{warning <'Multi will not function for Sectors that span multiple XTS tracks'>}    
FUNCTION_BLOCK FB_SingularTrackSector
VAR_INPUT
	PlanarTrackIndex				: E_TrackNum := E_TrackNum.Small;
END_VAR
VAR_IN_OUT
	refPlanarTracks					: ARRAY[*] OF ST_PlanarTrackConfig; //NOTE ref array is 0-based!
END_VAR                     		
VAR                             	
	InitDone						: BOOL;
	stSectorConfig					: ST_SectorConfig;
	LowerBoundPlanarTrackConfig		: DINT;
	UpperBoundPlanarTrackConfig		: DINT;
	refXtsMover						: Tc3_XTS_Utility.ST_PositionInfo;
	refPlanarMover					: MoverSort;
	stTrackSectorStatus				: ST_SectorStatus;
END_VAR

IF UpperBoundPlanarTrackConfig = 0 THEN
	_M_Init();
ELSE
	InitDone	:= TRUE;
END_IF

IF InitDone THEN
	_M_UpdateSectorStatus();
END_IF

METHOD PRIVATE _M_Init
LowerBoundPlanarTrackConfig	:= LOWER_BOUND(refPlanarTracks,1);
UpperBoundPlanarTrackConfig	:= UPPER_BOUND(refPlanarTracks,1);
END_METHOD

METHOD PROTECTED _M_IsOnPlanarSector : BOOL
//note refPlanarTracks ARRAY is 0-based!
IF ADR(refPlanarTracks[(PlanarTrackIndex-1)]) <> Tc3_Module.NULL THEN
	_M_IsOnPlanarSector	:= (refPlanarMover.TrackID = refPlanarTracks[(PlanarTrackIndex-1)].MCTrack.TrackOID) 
							AND IsBetween(value := refPlanarMover.MoverPos, 
												minV := stSectorConfig.TrackSectorStartPosn, 
												maxV := stSectorConfig.TrackSectorEndPosn);
END_IF
END_METHOD

METHOD PROTECTED _M_IsOnXtsSector : BOOL
_M_IsOnXtsSector	:= ((refXtsMover.nTrackObjectid = stSectorConfig.ObjectId) OR
											(refXtsMover.nPartObjectid = stSectorConfig.ObjectId)) AND
											(IsBetween(value := refXtsMover.fPartPosition, 
											minV := stSectorConfig.PartSectorStartPosn, 
											maxV := stSectorConfig.PartSectorEndPosn) OR
											IsBetween(value := refXtsMover.fTrackPosition, 
											minV := stSectorConfig.TrackSectorStartPosn, 
											maxV := stSectorConfig.TrackSectorEndPosn));
END_METHOD

METHOD PROTECTED _M_UpdateSectorStatus
stTrackSectorStatus.MoverIsOnSector	:= _M_IsOnXtsSector() OR _M_IsOnPlanarSector();

stTrackSectorStatus.MoverEnteredSector(CLK := stTrackSectorStatus.MoverIsOnSector);
stTrackSectorStatus.MoverExitedSector(CLK := stTrackSectorStatus.MoverIsOnSector);
END_METHOD

PROPERTY P_PlanarMover : REFERENCE TO MoverSort
GET
P_PlanarMover	REF= refPlanarMover;
END_GET
END_PROPERTY

PROPERTY P_SectorStatus : REFERENCE TO ST_SectorStatus
GET
P_SectorStatus	REF= stTrackSectorStatus;
END_GET
END_PROPERTY

PROPERTY P_TrackSectorConfig : REFERENCE TO ST_SectorConfig
GET
P_TrackSectorConfig REF= stSectorConfig;
END_GET
END_PROPERTY

PROPERTY P_XtsPositionInfo : REFERENCE TO Tc3_XTS_Utility.ST_PositionInfo
GET
P_XtsPositionInfo REF= refXtsMover;
END_GET
END_PROPERTY

END_FUNCTION_BLOCK

(* stored: Version 1.1.0.1
   POU FB_SingularTrackSector: Id {454c8ee6-eb93-03bb-3d09-d82885cc2db0}, SpecialFunc None
   Method _M_Init: Id {ef455004-cd91-0816-3ac9-eb75e5eaacf7}
   Method _M_IsOnPlanarSector: Id {801ce463-9c2b-0c61-1ed8-bdb6b24d5f35}
   Method _M_IsOnXtsSector: Id {6fb38ca4-6b76-0afd-297f-a5f43cfa3834}
   Method _M_UpdateSectorStatus: Id {3dbda7bd-d78d-0797-197a-6bd81167f773}
   Property P_PlanarMover: Id {c0ac9430-b382-04fd-3b6a-1962bd5a1c7e}
   Get Get: Id {804e0c8f-06ff-09a3-09d5-b11c0f048c58}
   Property P_SectorStatus: Id {5f8e870d-e32a-0163-2da9-1a6a40e1a497}
   Get Get: Id {de3ffc99-936a-0b5d-0ea1-4e9664bc445a}
   Property P_TrackSectorConfig: Id {5b7ff01c-1c59-02c5-1dcb-4c860620dc5f}
   Get Get: Id {6f251efa-6799-0ba7-38f2-aa9f1e2ed41e}
   Property P_XtsPositionInfo: Id {d96f07f7-f866-0c16-0900-c47c81882126}
   Get Get: Id {ae45bb6f-f61b-08ea-11d8-d62f8182115f} *)
